Yaskawa INFORM job: UPDATE_X_Y_Z.JBI

/JOB
//NAME UPDATE_X_Y_Z
///FOLDERNAME FOLDER001
//POS
///NPOS 0,0,0,0,0,0
//INST
///DATE 2025/10/02 15:23
///ATTR SC,RW
///GROUP1 RB1
NOP
PAUSE
CALL JOB:LOAD_BOTTOM_END_XYZ
CALL JOB:LOAD_TOP_START_XYZ
CALL JOB:LOAD_TOP_END_XYZ
CALL JOB:LOAD_BOTTOM_START_XYZ
END
